PROGRAM MAIN_test
VAR
	Motion_1	AT %I* 	: BOOL;
	Motion_2 	AT %I*	: BOOL;
	Relay_1 	AT %Q*	: BOOL;
	Relay_2 	AT %Q*	: BOOL;	
	vDruk_1				: BOOL;
	vDruk_2				: BOOL;	
	Druk_1		AT %I*	: BOOL;
	Druk_2		AT %I*	: BOOL;	
	LDR_1		AT %I* 	: INT;
	LDR_2		AT %I* 	: INT;
	LDR_3		AT %I* 	: INT;
	LDR_4		AT %I* 	: INT;
	
	TOF1			: TOF;
	F_TRIG1			: F_Trig;
	
	lichten_1		: lichten;
	lichten_2		: lichten;
	TOF2, TOF3		: TOF;
	F_TOF2, F_TOF3	: F_Trig;

	Inschakelen_1	: BOOL;
	ENABLE			: BOOL;
	TON1			: TON;
	
	automatic_1: automatic;
	automatic_2: automatic;
	auto_ON : BOOL;
END_VAR

automatic_1(	LDR1:= LDR_1, LDR2:= LDR_2, LDR_threshold:= 500, motion:= Motion_1 );
automatic_2(	LDR1:= LDR_3, LDR2:= LDR_4, LDR_threshold:= 500, motion:= Motion_2 );



IF druk_2 THEN auto_ON := NOT auto_ON; END_IF
				
IF auto_ON THEN
	lichten_1.ON:= automatic_1.ON;
	lichten_1.OFF:= automatic_1.OFF;
	lichten_2.ON:= automatic_2.ON;
	lichten_2.OFF := automatic_2.OFF;
ELSE
	lichten_1.ON:= FALSE;
	lichten_1.OFF:= FALSE;
	lichten_2.ON:= FALSE;
	lichten_2.OFF := FALSE;
END_IF
				
lichten_1(	toggle:= vDruk_1 OR Druk_1, 
			 Q=> Relay_1 );

lichten_2(	toggle:= vDruk_2 OR Druk_1, 
			ON:= automatic_2.ON, OFF:= automatic_2.OFF, Q=> Relay_2 );
			
beamer();

END_PROGRAM

(* stored: Version 1.1.0.1, ProductVersion 3.1.4022.12
   POU MAIN_test: Id {4011f441-4cc2-4873-9837-bdd0c0d42fbb}, SpecialFunc None *)
